(* CODESYS project Untitled1.project

Project tree, tasks and I/O mapping:
  Device : CODESYS Control Win V3, 3S - Smart Software Solutions GmbH, order no. 305021, version 3.5.11.30
    application Application
      libraries: Standard, * (System)
      task MainTask (cyclic, interval t#20ms, priority 1) calls PLC_PRG
      program PLC_PRG [ST]
      Symbols
*)

// Device/Application/PLC_PRG
PROGRAM PLC_PRG
VAR
	DELAY:BOOL;
	DELAY2:BOOL;
	//TIMERS
	TIMER: TON;
	TIMER2: TON;
	//BOTOES
	START_BUTTON: BOOL := 0;
	RESET: BOOL;
	//SENSORES
	VISION_SENSOR: ARRAY[1..4] OF BOOL;
	REFLECTIVE1: BOOL := 0;
	REFLECTIVE2: BOOL := 0;
	//ATUADORES
	POSITIONER1: BOOL := 0;
	POSITIONER2: BOOL := 0;
	CINZA: BOOL;
	VERDE: BOOL;
	AZUL: BOOL;
	EMITTER_PART: INT;
	EMIT: BOOL := 0;
	TRANSPORTADORA: BOOL := 0;
	TRANSPORTADORA2: BOOL := 0;
	//TWO-AXIS PICK & PLACE
	Z: REAL := 0;
	X: REAL := 1.1;
	Y: REAL := 0;
	GRAB: BOOL := 0;
	DETECTING: BOOL;
	ROTATINGccw: BOOL;
	//AUXILIARES
	PROGRESS_FLAG: WORD := 0;
	GRAB_FLAG: BOOL;
END_VAR

TIMER(IN:= DELAY, PT:= T#1S);
TIMER2(IN:= DELAY2, PT:= T#1S);
//RESET
IF RESET THEN
	Z := 0;
	X := 1.1;
	Y := 0;
	GRAB := 0;
	TRANSPORTADORA := 0;
	TRANSPORTADORA2 := 0;
	EMIT := FALSE;
	PROGRESS_FLAG := 0;
	GRAB_FLAG := 0;
	DELAY := 0;
	DELAY2 := 0;
	POSITIONER1 := 0;
	POSITIONER2 := 0;
	RESET := 0;
END_IF

//CONTROLANDO ESTEIRA
IF START_BUTTON AND PROGRESS_FLAG < 2 THEN
	TRANSPORTADORA := TRUE;
ELSE 
	TRANSPORTADORA := FALSE;
END_IF

//USANDO SENSOR PRA DETECTAR COR DE OBTEJO
IF (VISION_SENSOR[1] AND VISION_SENSOR[2]) THEN
	EMITTER_PART := 1024; TRANSPORTADORA2 := 1; CINZA := FALSE; VERDE := FALSE; AZUL := TRUE; //AZUL
	EMIT := TRUE;
	DELAY := TRUE;
	
ELSIF VISION_SENSOR[1] THEN
	EMITTER_PART := 4096; TRANSPORTADORA2 := 1; CINZA := TRUE; VERDE := FALSE; AZUL := FALSE; //CINZA
	EMIT := TRUE;
	DELAY := TRUE;
	
ELSIF VISION_SENSOR[3] THEN
	EMITTER_PART := 2048; TRANSPORTADORA2 := 1; CINZA := FALSE; VERDE := TRUE; AZUL := FALSE; //VERDE
	EMIT := TRUE;
	DELAY := TRUE;
END_IF

IF TIMER.Q THEN
	EMIT := FALSE;
	DELAY := FALSE;
END_IF

//CONTROLANDO PICK & PLACE
//PROGRESS = 1
IF NOT REFLECTIVE2 THEN
	PROGRESS_FLAG := 1;
	DELAY2 := TRUE;
END_IF

//PROGRESS = 2
IF POSITIONER1 THEN
	DELAY2:=TRUE;
END_IF

//PROGRESS = 3
IF DETECTING AND NOT GRAB_FLAG THEN
//	GRAB := TRUE;
//	Z := 4;
//	X := 0;
	GRAB_FLAG := TRUE;
	DELAY2 := 1;
END_IF

//PROGRESS = 4
IF GRAB_FLAG AND NOT DELAY2 THEN
	DELAY2 := TRUE;
END_IF

//PROGRESS = 5
IF PROGRESS_FLAG = 6 THEN
	DELAY2 := TRUE;
END_IF

IF Z = 3 THEN
	DELAY := TRUE;
END_IF

IF TIMER2.Q THEN
	DELAY2 := FALSE;
	IF PROGRESS_FLAG = 8 THEN
		GRAB := FALSE;	
		RESET := 1;
	
	ELSIF PROGRESS_FLAG = 7 THEN
		Y := 10;
		PROGRESS_FLAG := 8;
		
	ELSIF PROGRESS_FLAG = 6 THEN
		Z := 3;
		PROGRESS_FLAG := 7;
		
	ELSIF PROGRESS_FLAG = 5 THEN
		Z := 8.2;
		PROGRESS_FLAG := 6;
	
	ELSIF PROGRESS_FLAG = 4 THEN
		X := 6.4;
		PROGRESS_FLAG := 5;
		
	ELSIF PROGRESS_FLAG = 3 THEN
		Z := 3;
		PROGRESS_FLAG := 4;
		
	ELSIF PROGRESS_FLAG = 2 THEN
		POSITIONER1 := FALSE;
		POSITIONER2 := FALSE;
		TRANSPORTADORA2 := FALSE;
		GRAB := TRUE;
		Z := 8.2;
		PROGRESS_FLAG := 3;
		
	ELSIF PROGRESS_FLAG = 1 THEN
		POSITIONER1 := TRUE;
		POSITIONER2 := TRUE;
		PROGRESS_FLAG := 2;
	END_IF
END_IF

END_PROGRAM
